RoboDK station: New Station objects.rdk

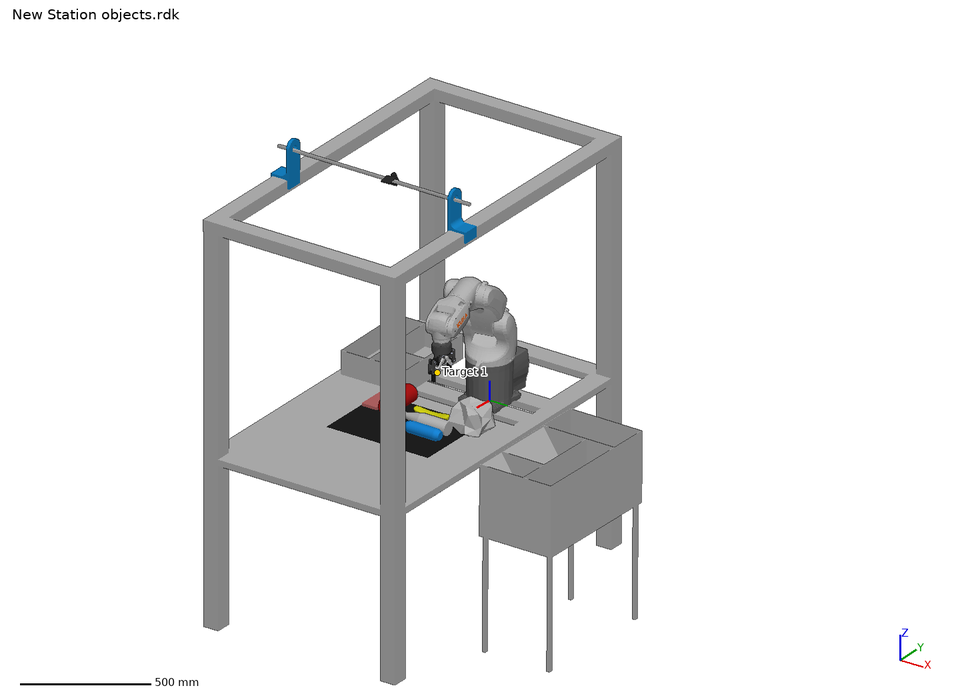
[picture v0: the station drawn from its stored meshes, robots at their saved joint values, targets as dots, program paths as lines]
Station New Station objects. Poses are relative to the parent item; angles as X-Y-Z fixed-axis rotations.
  - object  at (0, 0, 0) mm, size 107739.4 x 3125.1 x 1726.8 mm, geometry from  v2.stl
    - object  at (683.14, 692.28, 126.23) mm, size 11160.4 x 232.2 x 223 mm, geometry from 2 v1.stl
  - frame KUKA KR 3 R540 Base at (621.06, 1018.74, 14.92) mm, rotated rx 0 ry 0 rz -90.32 deg
    - robot KUKA KR 3 R540: 6 axes, payload 3 kg, reach 541 mm, repeatability 0.02 mm, weight 26 kg
        modified DH rows (alpha deg, a mm, theta deg, d mm): 0, 0, 0, 345; -90, 20, 0, 0; 0, 260, -90, 0; -90, 20, 0, 260; 90, 0, 0, 0; -90, 0, 180, 75
        joint limits [-170, -170, -110, -175, -120, -350] to [170, 50, 155, 175, 120, 350]; home [0, -90, 90, 0, 0, 0]; saved at [-11.47, -48.056, 56.732, 0, 81.325, -11.47]
      - tool Gripper RobotiQ 85 Opened, TCP at (0, -20, 130) mm, size 147.4 x 146.8 x 75 mm
    - target Target 1 (Cartesian target) at (444.76, 70.24, 313.94) mm, rotated rx 180 ry 0 rz -180 deg; joints [-11.47, -48.056, 56.732, 0, 81.325, -11.47] of KUKA KR 3 R540
  - object  at (331.87, 880.57, 17.64) mm, rotated rx 90 ry 0 rz -179.22 deg, size 304 x 104 x 379 mm, geometry from  v2.stl
  - object banana v1 at (592.07, 728.63, 14.46) mm, size 159.5 x 33.3 x 40.6 mm, geometry from banana v1.stl
  - object bank v1 at (381.05, 838.6, 91) mm, rotated rx 89.94 ry 0 rz 0 deg, size 76.9 x 76.9 x 170.3 mm, geometry from bank v1.stl
  - object botlle v1 at (672.59, 696.49, 47.16) mm, rotated rx 0 ry -89.42 rz 0 deg, size 60 x 60 x 252.8 mm, geometry from botlle v1.stl
  - object money v2 at (253.2, 851.32, 17.5) mm, size 69 x 157 x 12 mm, geometry from money v2.stl
  - object  at (679.59, 649.46, 41.97) mm, rotated rx 0 ry -89.61 rz 0 deg, size 49.9 x 49.9 x 188.1 mm, geometry from  v1.stl
  - object  at (890.83, 562.44, -299.52) mm, rotated rx 90 ry 0.43 rz 89.84 deg, size 604 x 794 x 334 mm, geometry from  v2.stl
  - object  at (272.61, 494.92, 15.5) mm, size 470 x 350 x 2 mm, geometry from  v1.stl
  - object  at (899.5, 462.71, 1015.05) mm, rotated rx 0 ry 0 rz 90.49 deg, size 72 x 85 x 200 mm, geometry from  v1.stl
  - object  at (-7.48, 532.19, 1016.27) mm, rotated rx 0 ry 0 rz -89.43 deg, size 72 x 85 x 200 mm, geometry from  v1.stl
  - object sick_for_cam v1 at (70.45, 498.74, 1125.41) mm, rotated rx 0 ry 0 rz -0.08 deg, size 895 x 10 x 10 mm, geometry from sick_for_cam v1.stl
  - object Cam1 v1 at (542.36, 504.65, 1137.85) mm, rotated rx -9.12 ry 0.26 rz -178.35 deg, size 40 x 74.5 x 42.3 mm, geometry from Cam1 v1.stl
  - object Cam1 fake at (516.75, 520.95, 1113.15) mm, rotated rx -178.74 ry -1.79 rz -0.04 deg, size 53 x 116 x 38 mm, geometry from Cam2D_SICK_VSPP_5F2113.sld
